// TwinCAT 3 PLC project PLc1
// ProgramVersion: 3.1.4023.0
// libraries:
//   Tc2_DALI, * (Beckhoff Automation GmbH)
//   Tc2_Standard, * (Beckhoff Automation GmbH)
//   Tc2_System, * (Beckhoff Automation GmbH)
//   Tc3_Database, * (Beckhoff Automation GmbH)
//   Tc3_EventLogger, * (Beckhoff Automation GmbH)
//   Tc3_Module, * (Beckhoff Automation GmbH)
// project tree:
//   DUTs/PLC_Expert/ E_Commands.TcDUT, E_DataSets.TcDUT, E_PLCDBState.TcDUT, ST_DB.TcDUT
//   DUTs/SQL_Expert/ ST_ResultEvent.TcDUT, ST_Select.TcDUT
//   / PlcTask.TcTTO
//   POUs/ MAIN.TcPOU, P_InfluxTEST.TcPOU, P_PLCExpert_AutoLog.TcPOU, P_PLCExpert_Independent_FBs.TcPOU, P_SQLExpert_DataRet.TcPOU, P_SQLExpert_NoDataRet.TcPOU
// real-time tasks:
//   TASK PlcTask: cycle T#10ms, priority 20, ADS port 350

CONFIGURATION PLc1
    RESOURCE PLC ON TwinCAT3
        TASK PlcTask(INTERVAL := T#10ms, PRIORITY := 20);
        PROGRAM MAIN WITH PlcTask : MAIN;
    END_RESOURCE
END_CONFIGURATION

// ---- DUTs/PLC_Expert/E_Commands.TcDUT
//{attribute 'qualified_only'}
{attribute 'strict'}
TYPE E_Commands :
(
	InsertIntoTable	 	:= 20,
	ClearTable 			:= 21,
	ReadAllfromTable	:= 22,
	CustomReadfromTable	:= 23,
	DropTable			:= 24
);
END_TYPE

// ---- DUTs/PLC_Expert/E_DataSets.TcDUT
//{attribute 'qualified_only'}
{attribute 'strict'}
TYPE E_DataSets :
(
	DataSet1 := 10,
	DataSet2 := 11,
	DataSet3 := 12
);
END_TYPE

// ---- DUTs/PLC_Expert/E_PLCDBState.TcDUT
//{attribute 'qualified_only'}
{attribute 'strict'}
TYPE E_PLCDBState :
(
	Wait 				:= 0,
	WriteData			:= 1,
	ReadData			:= 2,
	RunCMDCommand		:= 3,
	AutoLog				:= 4,
	CreateTable			:= 5,
	EventHandling		:= 9
);
END_TYPE

// ---- DUTs/PLC_Expert/ST_DB.TcDUT
TYPE ST_DB :
STRUCT
	ID			: LINT;
	Timestamp	: DT;
	Name		: STRING;
	Value		: LREAL;
END_STRUCT
END_TYPE

// ---- DUTs/SQL_Expert/ST_ResultEvent.TcDUT
TYPE ST_ResultEvent :
STRUCT
	gEventClass 			: 	GUID;
	wsEventClassDisplayName : 	WSTRING(255);
	udiEventId				: 	UDINT;
	eSeverity 				: 	TcEventSeverity;
	sSourcePath				:	T_MaxString;
	wsText					:	WSTRING(255);
END_STRUCT
END_TYPE

// ---- DUTs/SQL_Expert/ST_Select.TcDUT
TYPE ST_Select :
STRUCT
	ID: LINT;
	Timestamp: DT;
	Name: STRING(80);
	Value: LREAL;
END_STRUCT
END_TYPE

// ---- POUs/MAIN.TcPOU
PROGRAM MAIN
VAR
	rTemp					: REAL;
	rVar					: REAL;
	rVariablePLC			: REAL;
END_VAR

P_PLCExpert_AutoLog();
//P_PLCExpert_Independent_FBs();
//P_SQLExpert_NoDataRet();
//P_SQLExpert_DataRet();
//P_InfluxTEST();

END_PROGRAM

// ---- POUs/P_PLCExpert_AutoLog.TcPOU
PROGRAM P_PLCExpert_AutoLog
VAR
	
	fbPLCDBAutoLog  			: FB_PLCDBAutoLogEvt (sNetID:='', tTimeout := T#5S);						// PLCDBAutoLogEvt fb instance
	ipTcResult					: Tc3_Database.I_TcMessage;	
    aAutologGrpStatus 			: ARRAY[0..MAX_CONFIGURATIONS] OF ST_AutoLogGrpStatus;
	
	// Zmienne konfigurowalne przez użytkownika
	bRun						: BOOL;																		// TRUE AutoLog Start
	bStop						: BOOL;																		// TRUE AutoLog Stop
	tAutoLogStatusCheckCycle	: TIME 														:= T#3S;		// Okres pobierania statusu grupy auto logowania
	
END_VAR

IF bRun AND_THEN fbPLCDBAutoLog.Start() THEN						// Start grupy AutoLog za pomocą bRun
	bRun := FALSE;
END_IF

fbPLCDBAutoLog.Status(												// Pobranie infromacji o statusie grupy AutoLog
						tAutoLogStatusCheckCycle, 
						ADR(fbPLCDBAutoLog.bError), 
						ADR(aAutologGrpStatus), 
						SIZEOF(aAutologGrpStatus));

IF bStop AND NOT bRun AND_THEN fbPLCDBAutoLog.Stop() THEN			// Stop grupy AutoLog za pomocą bStop
	bStop := FALSE;
END_IF

IF NOT fbPLCDBAutoLog.bBusy THEN									// Zapisanie do struktury informacji o zwracanych przez blok funkcyjny danych
	ipTcResult := fbPLCDBAutoLog.ipTcResult;	
END_IF

END_PROGRAM

// ---- POUs/P_InfluxTEST.TcPOU
PROGRAM P_InfluxTEST
VAR
	rand 	: DRAND;							// Instance of DRAND function block
    nrand	: LREAL;			
	fValue1	: LREAL;
	fValue2	: LREAL;
	fValue3	: LREAL;
END_VAR

rand();
nrand := rand.Num;
fValue1 := 240.328 + 10 * nrand;
fValue2 := 7.3292 + nrand;
fValue3 := 1113.1975 + 50 * nrand;

END_PROGRAM

// ---- POUs/P_PLCExpert_Independent_FBs.TcPOU
PROGRAM P_PLCExpert_Independent_FBs
VAR																												
																
	fbPLCDBWrite	: FB_PLCDBWriteEvt(sNetID:='', tTimeout:=T#5S);								
	fbPLCDBRead		: FB_PLCDBReadEvt(sNetID:='', tTimeout:=T#5S);								
	fbPLCDBCmd		: FB_PLCDBCmdEvt(sNetID := '', tTimeout := T#5S);                           
	fbPLCDBAutoLog  : FB_PLCDBAutoLogEvt(sNetID:='', tTimeout := T#5S);							
	fbPLCDBCreate	: FB_PLCDBCreateEvt(sNetID:='', tTimeout := T#5S);
		
	arrColumns		: ARRAY[0..3] OF STRING[50] := ['ID', 'Timestamp', 'Name', 'Value'];		// Tablica zawierająca nazwy kolumn tabeli	
	arrData			: ARRAY[0..19] OF ST_DB;													// Tablica w której przechowywane będą dane z tabeli
	arrParameter	: ARRAY [0..3] OF ST_ExpParameter := [										// Tablica z parametrami tabeli
								(sParaName := 'id', 	nParaSize := 8,		eParaType := E_EXPPARAMETERTYPE.Int64), 
								(sParaName := 'time', 	nParaSize := 4, 	eParaType := E_EXPPARAMETERTYPE.DateTime),
								(sParaName := 'name', 	nParaSize := 81, 	eParaType := E_EXPPARAMETERTYPE.STRING_), 
								(sParaName := 'value', 	nParaSize := 8, 	eParaType := E_EXPPARAMETERTYPE.Double64)];
	
	ipTcResult		: Tc3_Database.I_TcMessage;													
	sSourceInfo		: Tc3_EventLogger.I_TcSourceInfo;											
	sEventClass		: Tc3_EventLogger.GUID;														
	eSeverity		: Tc3_EventLogger.TcEventSeverity;
	stEventEntry	: Tc3_EventLogger.TcEventEntry;	
	nEventID		: UDINT;																	// Event ID											

	sCommand		: STRING(1000);																// Będzie zawierać komendę SQL
	arrColumnInfo   : ARRAY [0..3] OF ST_ColumnInfo :=[											// Ustawienia nowej tabeli
								(sName := 'ID',			eType := E_ColumnType.BigInt, 	nLength := 8, 	sProperty := 'IDENTITY(1,1)'), 
								(sName := 'Timestamp', 	eType := E_ColumnType.DateTime, nLength := 8),
								(sName := 'Name', 		eType := E_ColumnType.NVarChar, nLength := 81),
								(sName := 'Value', 		eType := E_ColumnType.REAL_, 	nLength := 8)];											
	
	// Zmienne konfigurowalne przez użytkownika
	bRun			: BOOL;																		// Włączenie wszystkich grup autologowania
	hDBID			: UDINT 		:= 1;														// Numer bazy danych, na której chcemy wykonywać operacje
	sDBID			: STRING(50)	:= 'TESTtable';												// Nazwa bazy danych, na której chcemy wykonywać operacje
	eCommands		: E_Commands 	:= ReadAllfromTable;										// Wybranie komendy SQL
	ePLCDBState		: E_PLCDBState	:= Wait;													// Wybranie instrukcji, które mają być wykonane
	hAutoLogGroup	: UDINT			:= 1;														// Numer grupy autologowania, na której chcemy wykonywać operacje
	nRecords		: UDINT			:= 10;														// Liczba rekordów czytanych przez fbPLCDBCmd
	nInitialIndex	: UDINT			:= 0;														// Indeks pierwszego rekordu czytanego przez fbPLCDBCmd/fbPLCDBRead
	nRecordAmount	: UDINT			:= 20;														// Liczba rekordów, które zostaną przeczytane
	sOrderBy		: STRING(50)	:= 'ID';													// Wyznaczenie kolumny, według której dane bedą poukładane
	stDB			: ST_DB;																	// Struktura z wartościami zmiennych, które zostaną wpisane do tabeli za pomocą fbPLCDBWrite
END_VAR

CASE eCommands OF		//Wybranie realizowanej komendy SQL										
																
	InsertIntoTable:										  	
		sCommand := INSERT('INSERT INTO  (Timestamp, Name, Value) VALUES ( $'2018-01-31 14:59:27$', $'Temperature$', 21.3)', sDBID, 12);	
	ClearTable:													
		sCommand := INSERT('DELETE FROM ', sDBID, 12);       
	DropTable:													
		sCommand := INSERT('DROP TABLE ', sDBID, 11);        
																
		                                                        
	ReadAllfromTable: 											
		sCommand := INSERT('SELECT * FROM ', sDBID, 14);      
	CustomReadfromTable:										
		sCommand := INSERT('SELECT ID, Timestamp, Name, Value FROM  WHERE Value=21.3', sDBID, 39); 
		
END_CASE

CASE ePLCDBState OF												
	                                                            
	Wait:														
		;                                                       
		                                                        
	WriteData:			// Wpisanie danych do tabeli										
		fbPLCDBWrite.WriteStruct(								
		hDBID:= hDBID, 											
		sTableName:= sDBID, 									
		pRecord:= ADR(stDB), 															
		cbRecord:= SIZEOF(stDB), 								
		pColumnNames:= ADR(arrColumns), 						
		cbColumnNames:= SIZEOF(arrColumns));					
	                                                            
		IF NOT fbPLCDBWrite.bBusy THEN							
			ipTcResult := fbPLCDBWrite.ipTcResult;				
			IF NOT fbPLCDBWrite.bError THEN						
				ePLCDBState := ReadData;						
			ELSE												
				ePLCDBState := EventHandling;					
			END_IF
		END_IF
	
	ReadData:			// Odczytanie danych z tabeli										
		fbPLCDBRead.ReadStruct(									
		hDBID:= hDBID, 											
		sTableName:= sDBID, 									
		pColumnNames:= ADR(arrColumns), 						
		cbColumnNames:= SIZEOF(arrColumns), 					
		sOrderByColumn:= sOrderBy, 								
		eOrderType:= E_OrderType.ASC, 							
		nStartIndex:= nInitialIndex,	 						
		nRecordCount:= nRecordAmount, 							
		pData:= ADR(arrData), 									
		cbData:= SIZEOF(arrData));								
		                                                        
		IF NOT fbPLCDBRead.bBusy THEN							
		ipTcResult := fbPLCDBRead.ipTcResult;					
			IF NOT fbPLCDBRead.bError THEN						
				ePLCDBState := Wait;							
			ELSE												
				ePLCDBState := EventHandling;					
			END_IF
		END_IF
	
	RunCMDCommand: 		// Wykonanie komendy SQL										
	IF eCommands = InsertIntoTable OR eCommands = DropTable OR eCommands = ClearTable THEN
		fbPLCDBCmd.Execute(										
			hDBID:= hDBID, 										
			pExpression:= ADR(sCommand), 						
			cbExpression:= SIZEOF(sCommand), 					
			pData:= ADR(stDB), 									
			cbData:= SIZEOF(stDB), 								
			pParameter:= ADR(arrParameter), 					
			cbParameter:= SIZEOF(arrParameter));				
			                                                    
			IF NOT fbPLCDBCmd.bBusy THEN						
				ipTcResult := fbPLCDBRead.ipTcResult;			
				IF NOT fbPLCDBRead.bError THEN					
					ePLCDBState := ReadData;					
				ELSE											
					ePLCDBState := EventHandling;				
				END_IF
			END_IF
	ELSE														
		fbPLCDBCmd.ExecuteDataReturn(							
			hDBID:= hDBID, 										
			pExpression:= ADR(sCommand), 						
			cbExpression:= SIZEOF(sCommand), 					
			pData:= ADR(stDB), 									
			cbData:= SIZEOF(stDB), 								
			pParameter:= ADR(arrParameter), 					
			cbParameter:= SIZEOF(arrParameter), 				
			nStartIndex:= nInitialIndex, 						
			nRecordCount:= nRecordAmount, 						
			pReturnData:= ADR(arrData), 						
			cbReturnData:= SIZEOF(arrData), 					
			pRecords:= ADR(nRecords));							
			IF NOT fbPLCDBCmd.bBusy THEN						
				ipTcResult := fbPLCDBRead.ipTcResult;			
				IF NOT fbPLCDBRead.bError THEN					
					ePLCDBState := Wait;						
				ELSE											
					ePLCDBState := EventHandling;				
				END_IF
			END_IF
	END_IF	
			
	AutoLog:			// Jednokrotne zebranie wartości zmiennych zdefiniowanych w grupie auto logowania											
		fbPLCDBAutoLog.RunOnce(hAutologGrpID := hAutoLogGroup, bAll := bRun);
		IF NOT fbPLCDBAutoLog.bBusy THEN						
			ipTcResult := fbPLCDBAutoLog.ipTcResult;			
			IF NOT fbPLCDBAutoLog.bError THEN					
				ePLCDBState := ReadData;						
			ELSE												
				ePLCDBState := EventHandling;					
			END_IF
		END_IF
	
	CreateTable:		// Stworzenie nowej tabeli
		fbPLCDBCreate.Table(
				hDBID:= hDBID, 
				sTableName:= sDBID, 
				pTableCfg:= ADR(arrColumnInfo), 
				cbTableCfg:= SIZEOF(arrColumnInfo));
		IF NOT fbPLCDBCreate.bBusy THEN
			ipTcResult := fbPLCDBCreate.ipTcResult;
			IF NOT fbPLCDBCreate.bError THEN	
				ePLCDBState := wait;
			ELSE								
				ePLCDBState := EventHandling;
			END_IF
		END_IF
		
	EventHandling:		// Zebranie informacji o błędach									
		sSourceInfo := ipTcResult.ipSourceInfo;					
		sEventClass := ipTcResult.EventClass;					
		eSeverity 	:= ipTcResult.eSeverity;					
		nEventID	:= ipTcResult.nEventId;						
		stEventEntry:= ipTcResult.stEventEntry;					
	                                                            
		ePLCDBState := Wait;									
	
END_CASE

END_PROGRAM

// ---- POUs/P_SQLExpert_DataRet.TcPOU
PROGRAM P_SQLExpert_DataRet
//Program realizuje komendę SQL SELECT dla przykładowej tabeli.
VAR
	fbSQLDB					: 	FB_SQLDatabaseEvt(sNetID:='', tTimeout:=T#10S);
	fbSQLCmd 				: 	FB_SQLCommandEvt(sNetID:='', tTimeout:=T#10S);
	fbSQLResult				:	FB_SQLResultEvt(sNetID:='', tTimeout:=T#30S);
	iResult		 			:	Tc3_Database.I_TcMessage;						//Struktura w której zapisywane są dane o stanie komunikacji z bazą
	sQuery					: 	STRING(253);
	iState					:	INT;
	stSelect				: 	ST_Select;										//Struktura w której zapisywany jest wynik komendy SELECT
	sSqlCmdSelect			:	STRING						:= 'SELECT ID, Timestamp, Name, Value FROM  WHERE Value=21.3';	// Komenda SQL
				
	// Zmienne konfigurowalne przez użytkownika
	hDBID					:	UDINT 						:= 1;				//DBID bazy danych z którą się komunikujemy
	bRead					:	BOOL;
	udiStartIndex			:	UDINT						:= 0;				//Indeks od którego będą odczytywane rekordy
	udiRecordCount			:	UDINT						:= 1;				//Liczba odczytanych rekordów
	sTableName				:	STRING						:= 'TESTtable';		//Nazwa tabeli, na której wykonujemy komendę
	
	
END_VAR

CASE iState OF
	0: //bRead rozpoczyna program
		IF bRead THEN
			bRead := FALSE;
			iState := iState + 10;
		END_IF
		
	10: //Połączenie z bazą danych
		IF fbSQLDB.Connect(hDBID) THEN
			iResult := fbSQLDB.ipTcResult;
			IF fbSQLDB.bError THEN
				iState := 99;
			ELSE
				iState := iState + 10;
			END_IF
		END_IF 
		
	20: //Stworzenie komendy SQL - wstawienie do tabeli rekordu
		fbSQLDB.CreateCmd(pSQLCommand:= ADR(fbSQLCmd));
		IF NOT fbSQLDB.bBusy THEN
			iResult := fbSQLDB.ipTcResult;
			IF fbSQLDB.bError THEN
				iState := 99;
			ELSE
				iState := iState + 10;
				sQuery :=INSERT('SELECT ID, Timestamp, Name, Value FROM  WHERE Value=21.3', sTableName, 39);
			END_IF
		END_IF
		
	30: //Przygotowanie danych
		fbSQLCmd.ExecuteDataReturn(
									pSQLCmd := ADR(sQuery),
									cbSQLCmd := TO_UDINT(LEN(sQuery) + 1),
									pSQLDBResult := ADR(fbSQLResult));
		IF NOT fbSQLCmd.bBusy THEN
			iResult := fbSQLCmd.ipTcResult;
			IF fbSQLCmd.bError THEN
				iState := 99;
			ELSE
				 iState := iState + 10;
			END_IF
		END_IF

	40: //Umieszczenie danych w pamięci podręcznej
		fbSQLResult.Read(
				nStartIndex:= udiStartIndex, 
				nRecordCount:= udiRecordCount, 
				pData:= ADR(stSelect), 
				cbData:= SIZEOF(stSelect), 
				bWithVerifying:= FALSE , 
				bDataRelease:= TRUE);

		IF NOT fbSQLResult.bBusy THEN
			iResult := fbSQLResult.ipTcResult;
			IF fbSQLResult.bError THEN
				iState := 99;
			else
				iState := iState + 10;
			END_IF
		END_IF
		
	50: //Uwolnienie danych z pamięci podręcznej
		fbSQLResult.Release();
		IF NOT fbSQLResult.bBusy THEN
			iResult := fbSQLResult.ipTcResult;
			IF fbSQLResult.bError THEN
				iState := 99;
			else
				iState := iState + 10;
			END_IF
		END_IF
		
	60:	//Rozłączenie sie z bazą danych
		fbSQLDB.Disconnect();
		IF NOT fbSQLDB.bBusy THEN
			iResult := fbSQLDB.ipTcResult;
			IF fbSQLDB.bError THEN
				iState := 99;
			else
				iState := 0;
			END_IF
		END_IF
		
	99: // Error
		fbSQLDB.Disconnect();
		iState := 0;
END_CASE

END_PROGRAM

// ---- POUs/P_SQLExpert_NoDataRet.TcPOU
PROGRAM P_SQLExpert_NoDataRet
//Program wykonuje komendę SQL INSERT dla przykładowej tabeli. Jeśli tabela nie istnieje tworzy ją.
VAR
	fbSQLDB					: 	FB_SQLDatabaseEvt(sNetID:='', tTimeout:=T#10S);
	fbSQLCmd 				: 	FB_SQLCommandEvt(sNetID:='', tTimeout:=T#10S);
	fbSQLResult				:	FB_SQLResultEvt(sNetID:='', tTimeout:=T#30S);
	iResult		 			:	Tc3_Database.I_TcMessage;							//Struktura, w której zapisywane są dane o stanie komunikacji z bazą
	sQuery					: 	STRING(254);
	iState					:	INT;
	// Komenda tworząca tabelę, jeśli taka o podanej nazwie nie istnieje
	sSqlCmdCreateTable		:	STRING(254)				:= 'CREATE TABLE IF NOT EXISTS "" ("ID" INTEGER PRIMARY KEY AUTOINCREMENT NOT NULL, "Timestamp" DATETIME, "Name" VARCHAR(80), "Value" FLOAT)';
	// Komenda dodająca rekord do tabeli
	sSqlCmdInsertInto		:	STRING(254)				:= 'INSERT INTO  (Timestamp, Name, Value) VALUES ( $'2018-01-31 14:59:27$', $'Temperature$', 21.3)';
	
	
	// Zmienne konfigurowalne przez użytkownika
	sTableName				:	STRING					:= 'TESTtable'; 			//Nazwa tabeli, do której dodajemy rekordy
	hDBID					:	UDINT := 1;											//DBID bazy danych z którą się komunikujemy
	bInsert					:	BOOL;
END_VAR

CASE iState OF
	0:	//bInsert rozpoczyna program
		IF bInsert THEN
			bInsert := FALSE;
			iState := iState + 10;
		END_IF
		
	10:	//Połączenie z bazą danych
		IF fbSQLDB.Connect(hDBID) THEN
			iResult := fbSQLDB.ipTcResult;
			IF fbSQLDB.bError THEN
				iState := 99;
			ELSE
				iState := iState + 10;
			END_IF
		END_IF 
		
	20:	//Stworzenie komendy SQL - utworzenie tabeli jeśli nie istnieje
		fbSQLDB.CreateCmd(pSQLCommand := ADR(fbSQLCmd));
		IF NOT fbSQLDB.bBusy THEN
			iResult := fbSQLDB.ipTcResult;
			IF fbSQLDB.bError THEN
				iState := 99;
			ELSE
				iState := iState + 10;
				sQuery := INSERT(sSqlCmdCreateTable, sTableName, 28);
			END_IF
		END_IF
		
	30: //Przekazanie komendy i jej wykonanie
		fbSQLCmd.Execute(pSQLCmd := ADR(sQuery), cbSQLCmd := TO_UDINT(LEN(sQuery) + 1));
		IF NOT fbSQLCmd.bBusy THEN
			iResult := fbSQLCmd.ipTcResult;
			IF fbSQLCmd.bError THEN
				iState := 99;
			ELSE
				 iState := iState + 10;
			END_IF
		END_IF
		
	40:	//Stworzenie komendy SQL - wstawienie do tabeli rekordu
		fbSQLDB.CreateCmd(pSQLCommand := ADR(fbSQLCmd));
		IF NOT fbSQLDB.bBusy THEN
			iResult := fbSQLDB.ipTcResult;
			IF fbSQLDB.bError THEN
				iState := 99;
			ELSE
				iState := iState + 10;
				sQuery := INSERT(sSqlCmdInsertInto, sTableName, 12);
			END_IF
		END_IF
		
	50: //Przekazanie komendy i jej wykonanie
		fbSQLCmd.Execute(pSQLCmd := ADR(sQuery), cbSQLCmd := TO_UDINT(LEN(sQuery) + 1));
		IF NOT fbSQLCmd.bBusy THEN
			iResult := fbSQLCmd.ipTcResult;
			IF fbSQLCmd.bError THEN
				iState := 99;
			ELSE
				 iState := iState + 10;
			END_IF
		END_IF
		
	60:	//Rozłączenie się z bazą danych
		fbSQLDB.Disconnect();
		IF NOT fbSQLDB.bBusy THEN
			iResult := fbSQLDB.ipTcResult;
			IF fbSQLDB.bError THEN
				iState := 99;
			else
				iState := 0;
			END_IF
		END_IF
		
	99: // Error
		fbSQLDB.Disconnect();
		iState := 0;
END_CASE

END_PROGRAM
